FUNCTION_BLOCK EventLogger
VAR_INPUT
END_VAR
VAR_OUTPUT
END_VAR
VAR
END_VAR

END_FUNCTION_BLOCK

(* stored: Version 1.1.0.1, ProductVersion 3.1.4024.16
   POU EventLogger: Id {ce55a1a6-651b-4d1c-b136-d68617123420}, SpecialFunc None *)
